// SIMATIC S7-200 project (STEP 7-Micro/WIN), CPU 224XP REL 02.01

SYMBOL_TABLE USUARIO1
P_DERECHA        I0.0
P_IZQUIERDA      I0.1
P_PARO           I0.2
TERMICO          I0.4
M_DERECHA        Q0.0
LED_DERECHA      Q0.1
M_IZQUIERDA      Q0.2
LED_IZQUIERDA    Q0.3
LED_PAR0         Q0.4
AVERIA           Q0.5
END_SYMBOL_TABLE

SYMBOL_TABLE Símbolos S7-200
Primer_ciclo_ON  SM0.1    // ON sólo en el primer ciclo
END_SYMBOL_TABLE

ORGANIZATION_BLOCK PRINCIPAL:OB1
TITLE=COMENTARIOS DEL PROGRAMA
BEGIN
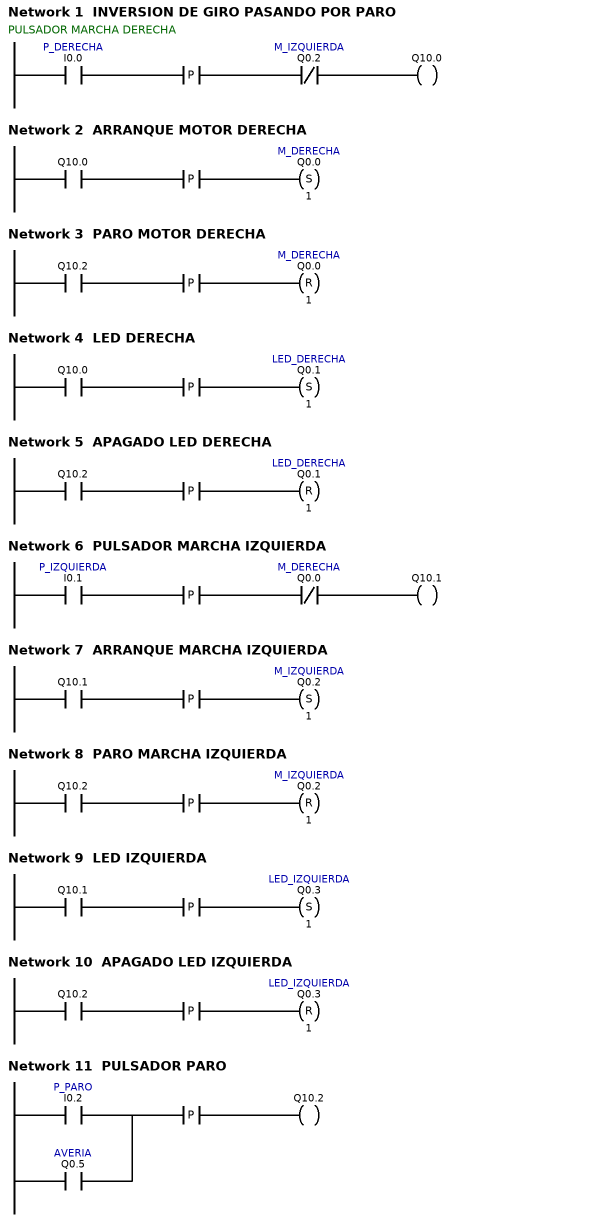
Network 1 // INVERSION DE GIRO PASANDO POR PARO
// PULSADOR MARCHA DERECHA 
LD     P_DERECHA:I0.0
EU
AN     M_IZQUIERDA:Q0.2
=      Q10.0
Network 2 // ARRANQUE MOTOR DERECHA 
LD     Q10.0
EU
S      M_DERECHA:Q0.0, 1
Network 3 // PARO MOTOR DERECHA
LD     Q10.2
EU
R      M_DERECHA:Q0.0, 1
Network 4 // LED DERECHA
LD     Q10.0
EU
S      LED_DERECHA:Q0.1, 1
Network 5 // APAGADO LED DERECHA
LD     Q10.2
EU
R      LED_DERECHA:Q0.1, 1
Network 6 // PULSADOR MARCHA IZQUIERDA
LD     P_IZQUIERDA:I0.1
EU
AN     M_DERECHA:Q0.0
=      Q10.1
Network 7 // ARRANQUE MARCHA IZQUIERDA
LD     Q10.1
EU
S      M_IZQUIERDA:Q0.2, 1
Network 8 // PARO MARCHA IZQUIERDA
LD     Q10.2
EU
R      M_IZQUIERDA:Q0.2, 1
Network 9 // LED IZQUIERDA 
LD     Q10.1
EU
S      LED_IZQUIERDA:Q0.3, 1
Network 10 // APAGADO LED IZQUIERDA
LD     Q10.2
EU
R      LED_IZQUIERDA:Q0.3, 1
Network 11 // PULSADOR PARO
LD     P_PARO:I0.2
O      AVERIA:Q0.5
EU
=      Q10.2
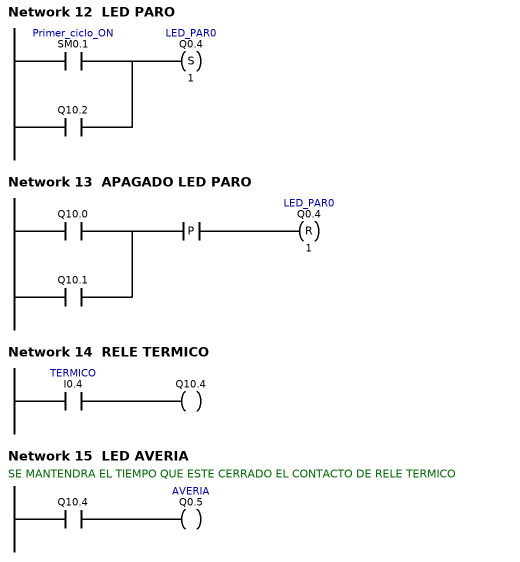
Network 12 // LED PARO
LD     Primer_ciclo_ON:SM0.1
O      Q10.2
S      LED_PAR0:Q0.4, 1
Network 13 // APAGADO LED PARO
LD     Q10.0
O      Q10.1
EU
R      LED_PAR0:Q0.4, 1
Network 14 // RELE TERMICO
LD     TERMICO:I0.4
=      Q10.4
Network 15 // LED AVERIA 
// SE MANTENDRA EL TIEMPO QUE ESTE CERRADO EL CONTACTO DE RELE TERMICO
LD     Q10.4
=      AVERIA:Q0.5
END_ORGANIZATION_BLOCK
